# EPICS autosave request: optics/opticsApp/Db/pf4bank_settings.req
$(P)$(H)debug$(B)
$(P)$(H)fPos$(B)
$(P)$(H)bank$(B)
$(P)$(H)bitFlag$(B)
$(P)$(H)status$(B)
$(P)$(H)f1$(B)
$(P)$(H)f2$(B)
$(P)$(H)f3$(B)
$(P)$(H)f4$(B)
$(P)$(H)Z1$(B)
$(P)$(H)Z2$(B)
$(P)$(H)Z3$(B)
$(P)$(H)Z4$(B)
$(P)$(H)Other1$(B)
$(P)$(H)Other2$(B)
$(P)$(H)Other3$(B)
$(P)$(H)Other4$(B)
